// TIA Portal V17 export
// export: Created 2024-09-02T12:50:34.0029074Z, ExportSetting WithDefaults, DisplayName Totally Integrated Automation Portal, DisplayVersion V17, DisplayName TIA Portal Openness, DisplayVersion V17, DisplayName TIA Portal Version Control Interface, DisplayVersion V17, DisplayName STEP 7 Professional, DisplayVersion V17, DisplayName STEP 7 Safety, DisplayVersion V17, DisplayName WinCC Professional, DisplayVersion V17
TYPE "TypeMobyVorgaben"
TITLE = moby addresses / Mobyadressen
// stored: IsFailsafeCompliant false
   STRUCT
      Kopiert { ExternalWritable := 'False'} : Bool;
      SchluesNr { ExternalWritable := 'False'} : Word;
      StationsNr { ExternalWritable := 'False'} : Int;
      PF { ExternalWritable := 'False'} : Array[1..8] of Bool;
      TAFaktiv { ExternalWritable := 'False'} : Array[1..8] of Bool;
   END_STRUCT;
END_TYPE
